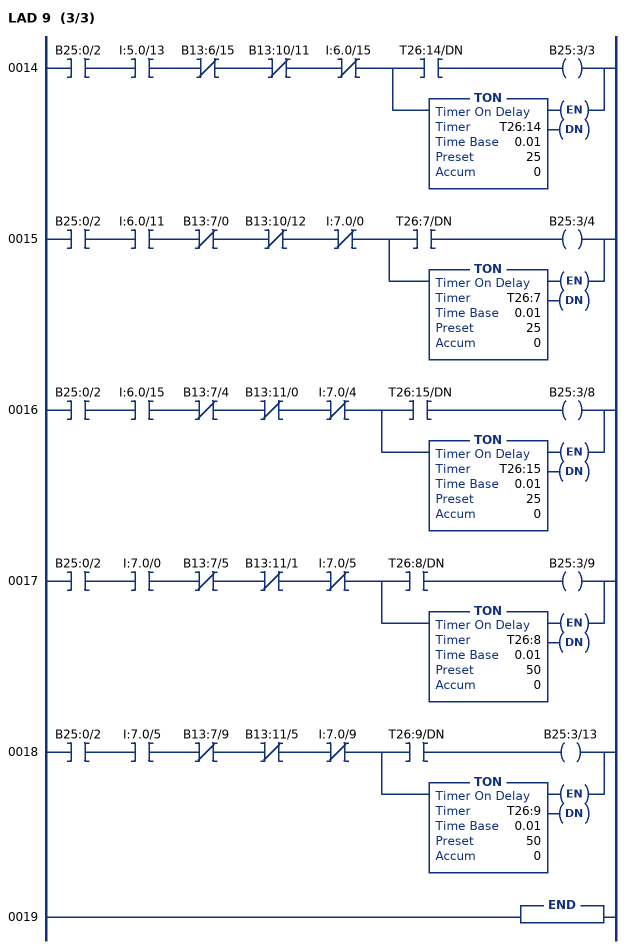
% Rung: 14 %
SOR XIC B25:0/2 XIC I:5.0/13 XIO B13:6/15 XIO B13:10/11 XIO I:6.0/15 BST XIC T26:14/DN OTE B25:3/3 NXB TON T26:14 0.01 25 0 BND EOR
% Rung: 15 %
SOR XIC B25:0/2 XIC I:6.0/11 XIO B13:7/0 XIO B13:10/12 XIO I:7.0/0 BST XIC T26:7/DN OTE B25:3/4 NXB TON T26:7 0.01 25 0 BND EOR
% Rung: 16 %
SOR XIC B25:0/2 XIC I:6.0/15 XIO B13:7/4 XIO B13:11/0 XIO I:7.0/4 BST XIC T26:15/DN OTE B25:3/8 NXB TON T26:15 0.01 25 0 BND EOR
% Rung: 17 %
SOR XIC B25:0/2 XIC I:7.0/0 XIO B13:7/5 XIO B13:11/1 XIO I:7.0/5 BST XIC T26:8/DN OTE B25:3/9 NXB TON T26:8 0.01 50 0 BND EOR
% Rung: 18 %
SOR XIC B25:0/2 XIC I:7.0/5 XIO B13:7/9 XIO B13:11/5 XIO I:7.0/9 BST XIC T26:9/DN OTE B25:3/13 NXB TON T26:9 0.01 50 0 BND EOR
% Rung: 19 %
SOR END EOR

LADDER 10
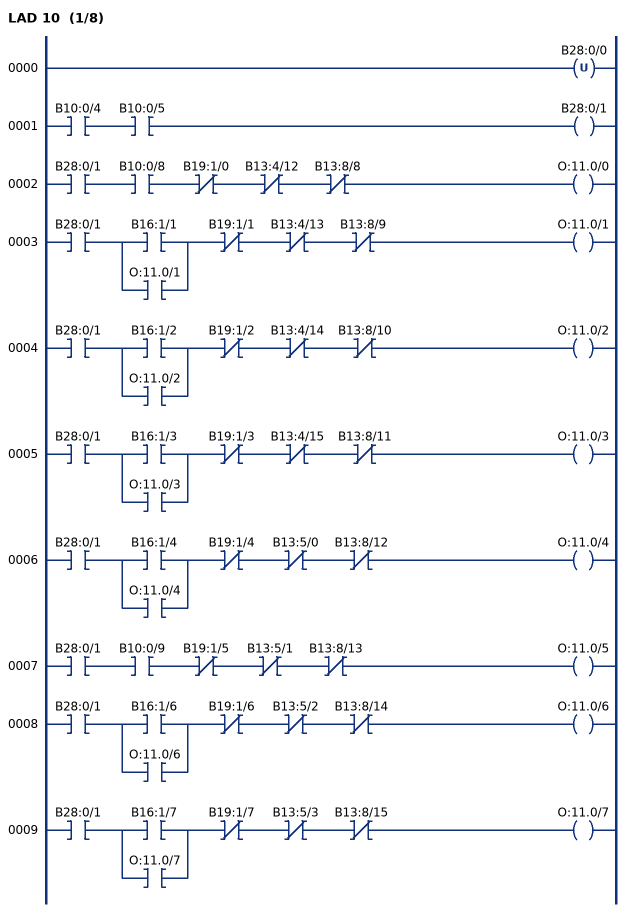
% Rung: 0 %
SOR OTU B28:0/0 EOR
% Rung: 1 %
SOR XIC B10:0/4 XIC B10:0/5 OTE B28:0/1 EOR
% Rung: 2 %
SOR XIC B28:0/1 XIC B10:0/8 XIO B19:1/0 XIO B13:4/12 XIO B13:8/8 OTE O:11.0/0 EOR
% Rung: 3 %
SOR XIC B28:0/1 BST XIC B16:1/1 NXB XIC O:11.0/1 BND XIO B19:1/1 XIO B13:4/13 XIO B13:8/9 OTE O:11.0/1 EOR
% Rung: 4 %
SOR XIC B28:0/1 BST XIC B16:1/2 NXB XIC O:11.0/2 BND XIO B19:1/2 XIO B13:4/14 XIO B13:8/10 OTE O:11.0/2 EOR
% Rung: 5 %
SOR XIC B28:0/1 BST XIC B16:1/3 NXB XIC O:11.0/3 BND XIO B19:1/3 XIO B13:4/15 XIO B13:8/11 OTE O:11.0/3 EOR
% Rung: 6 %
SOR XIC B28:0/1 BST XIC B16:1/4 NXB XIC O:11.0/4 BND XIO B19:1/4 XIO B13:5/0 XIO B13:8/12 OTE O:11.0/4 EOR
% Rung: 7 %
SOR XIC B28:0/1 XIC B10:0/9 XIO B19:1/5 XIO B13:5/1 XIO B13:8/13 OTE O:11.0/5 EOR
% Rung: 8 %
SOR XIC B28:0/1 BST XIC B16:1/6 NXB XIC O:11.0/6 BND XIO B19:1/6 XIO B13:5/2 XIO B13:8/14 OTE O:11.0/6 EOR
% Rung: 9 %
SOR XIC B28:0/1 BST XIC B16:1/7 NXB XIC O:11.0/7 BND XIO B19:1/7 XIO B13:5/3 XIO B13:8/15 OTE O:11.0/7 EOR

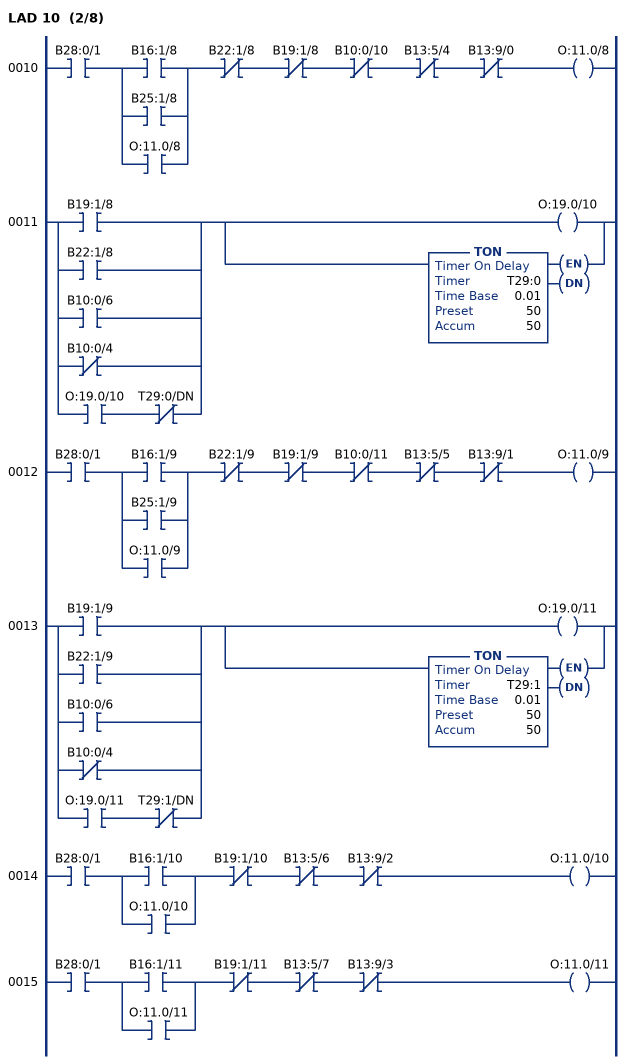
% Rung: 10 %
SOR XIC B28:0/1 BST XIC B16:1/8 NXB XIC B25:1/8 NXB XIC O:11.0/8 BND XIO B22:1/8 XIO B19:1/8 XIO B10:0/10 XIO B13:5/4 XIO B13:9/0 OTE O:11.0/8 EOR
% Rung: 11 %
SOR BST XIC B19:1/8 NXB XIC B22:1/8 NXB XIC B10:0/6 NXB XIO B10:0/4 NXB XIC O:19.0/10 XIO T29:0/DN BND BST OTE O:19.0/10 NXB TON T29:0 0.01 50 50 BND EOR
% Rung: 12 %
SOR XIC B28:0/1 BST XIC B16:1/9 NXB XIC B25:1/9 NXB XIC O:11.0/9 BND XIO B22:1/9 XIO B19:1/9 XIO B10:0/11 XIO B13:5/5 XIO B13:9/1 OTE O:11.0/9 EOR
% Rung: 13 %
SOR BST XIC B19:1/9 NXB XIC B22:1/9 NXB XIC B10:0/6 NXB XIO B10:0/4 NXB XIC O:19.0/11 XIO T29:1/DN BND BST OTE O:19.0/11 NXB TON T29:1 0.01 50 50 BND EOR
% Rung: 14 %
SOR XIC B28:0/1 BST XIC B16:1/10 NXB XIC O:11.0/10 BND XIO B19:1/10 XIO B13:5/6 XIO B13:9/2 OTE O:11.0/10 EOR
% Rung: 15 %
SOR XIC B28:0/1 BST XIC B16:1/11 NXB XIC O:11.0/11 BND XIO B19:1/11 XIO B13:5/7 XIO B13:9/3 OTE O:11.0/11 EOR

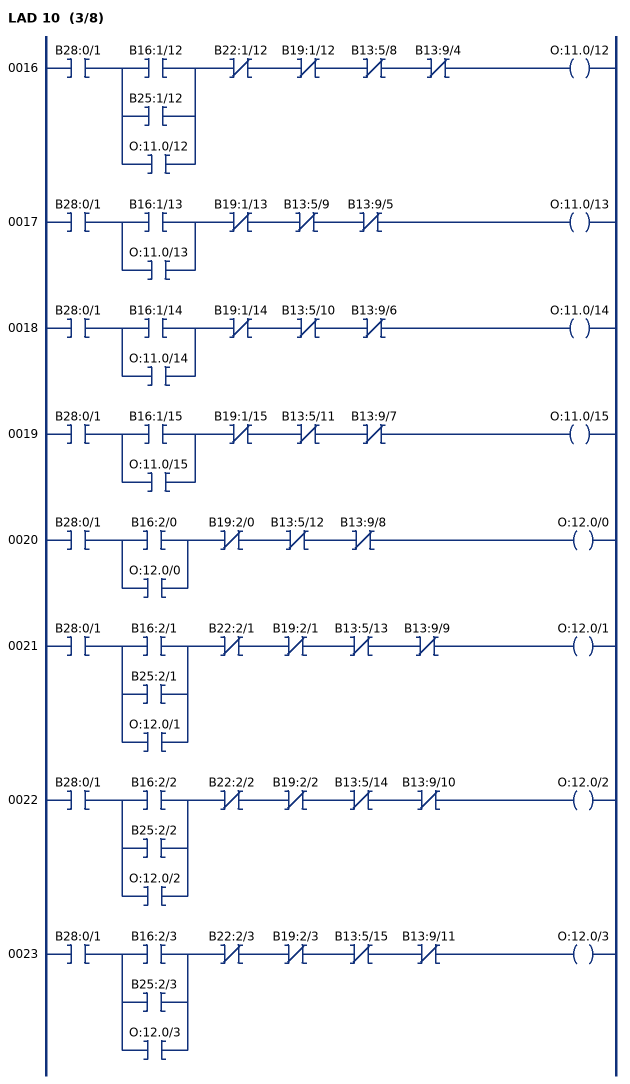
% Rung: 16 %
SOR XIC B28:0/1 BST XIC B16:1/12 NXB XIC B25:1/12 NXB XIC O:11.0/12 BND XIO B22:1/12 XIO B19:1/12 XIO B13:5/8 XIO B13:9/4 OTE O:11.0/12 EOR
% Rung: 17 %
SOR XIC B28:0/1 BST XIC B16:1/13 NXB XIC O:11.0/13 BND XIO B19:1/13 XIO B13:5/9 XIO B13:9/5 OTE O:11.0/13 EOR
% Rung: 18 %
SOR XIC B28:0/1 BST XIC B16:1/14 NXB XIC O:11.0/14 BND XIO B19:1/14 XIO B13:5/10 XIO B13:9/6 OTE O:11.0/14 EOR
% Rung: 19 %
SOR XIC B28:0/1 BST XIC B16:1/15 NXB XIC O:11.0/15 BND XIO B19:1/15 XIO B13:5/11 XIO B13:9/7 OTE O:11.0/15 EOR
% Rung: 20 %
SOR XIC B28:0/1 BST XIC B16:2/0 NXB XIC O:12.0/0 BND XIO B19:2/0 XIO B13:5/12 XIO B13:9/8 OTE O:12.0/0 EOR
% Rung: 21 %
SOR XIC B28:0/1 BST XIC B16:2/1 NXB XIC B25:2/1 NXB XIC O:12.0/1 BND XIO B22:2/1 XIO B19:2/1 XIO B13:5/13 XIO B13:9/9 OTE O:12.0/1 EOR
% Rung: 22 %
SOR XIC B28:0/1 BST XIC B16:2/2 NXB XIC B25:2/2 NXB XIC O:12.0/2 BND XIO B22:2/2 XIO B19:2/2 XIO B13:5/14 XIO B13:9/10 OTE O:12.0/2 EOR
% Rung: 23 %
SOR XIC B28:0/1 BST XIC B16:2/3 NXB XIC B25:2/3 NXB XIC O:12.0/3 BND XIO B22:2/3 XIO B19:2/3 XIO B13:5/15 XIO B13:9/11 OTE O:12.0/3 EOR

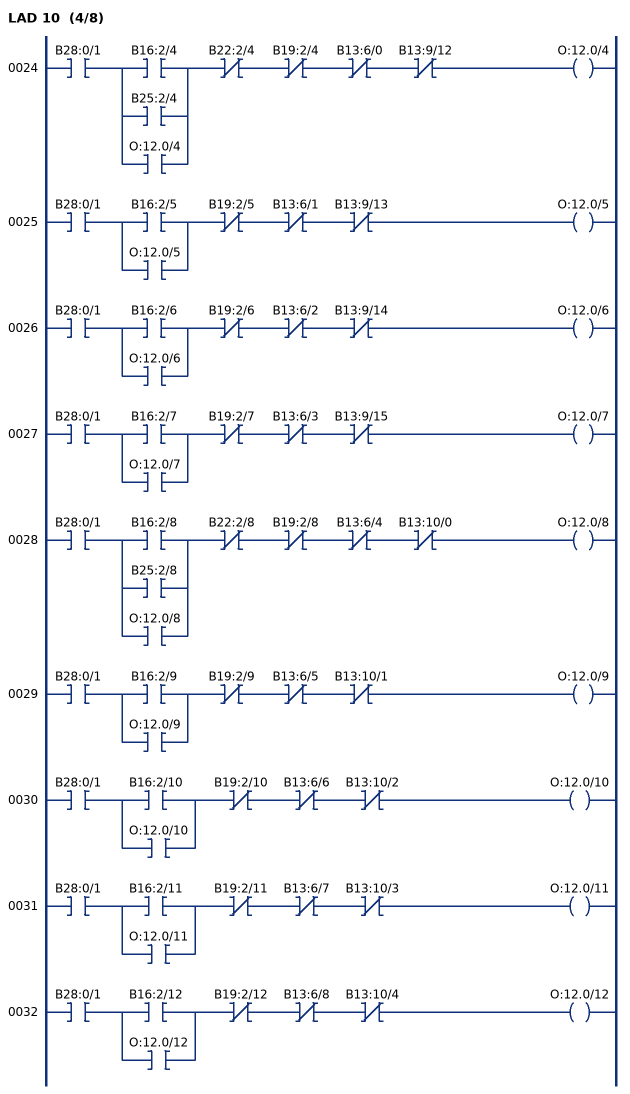
% Rung: 24 %
SOR XIC B28:0/1 BST XIC B16:2/4 NXB XIC B25:2/4 NXB XIC O:12.0/4 BND XIO B22:2/4 XIO B19:2/4 XIO B13:6/0 XIO B13:9/12 OTE O:12.0/4 EOR
% Rung: 25 %
SOR XIC B28:0/1 BST XIC B16:2/5 NXB XIC O:12.0/5 BND XIO B19:2/5 XIO B13:6/1 XIO B13:9/13 OTE O:12.0/5 EOR
% Rung: 26 %
SOR XIC B28:0/1 BST XIC B16:2/6 NXB XIC O:12.0/6 BND XIO B19:2/6 XIO B13:6/2 XIO B13:9/14 OTE O:12.0/6 EOR
% Rung: 27 %
SOR XIC B28:0/1 BST XIC B16:2/7 NXB XIC O:12.0/7 BND XIO B19:2/7 XIO B13:6/3 XIO B13:9/15 OTE O:12.0/7 EOR
% Rung: 28 %
SOR XIC B28:0/1 BST XIC B16:2/8 NXB XIC B25:2/8 NXB XIC O:12.0/8 BND XIO B22:2/8 XIO B19:2/8 XIO B13:6/4 XIO B13:10/0 OTE O:12.0/8 EOR
% Rung: 29 %
SOR XIC B28:0/1 BST XIC B16:2/9 NXB XIC O:12.0/9 BND XIO B19:2/9 XIO B13:6/5 XIO B13:10/1 OTE O:12.0/9 EOR
% Rung: 30 %
SOR XIC B28:0/1 BST XIC B16:2/10 NXB XIC O:12.0/10 BND XIO B19:2/10 XIO B13:6/6 XIO B13:10/2 OTE O:12.0/10 EOR
% Rung: 31 %
SOR XIC B28:0/1 BST XIC B16:2/11 NXB XIC O:12.0/11 BND XIO B19:2/11 XIO B13:6/7 XIO B13:10/3 OTE O:12.0/11 EOR
% Rung: 32 %
SOR XIC B28:0/1 BST XIC B16:2/12 NXB XIC O:12.0/12 BND XIO B19:2/12 XIO B13:6/8 XIO B13:10/4 OTE O:12.0/12 EOR

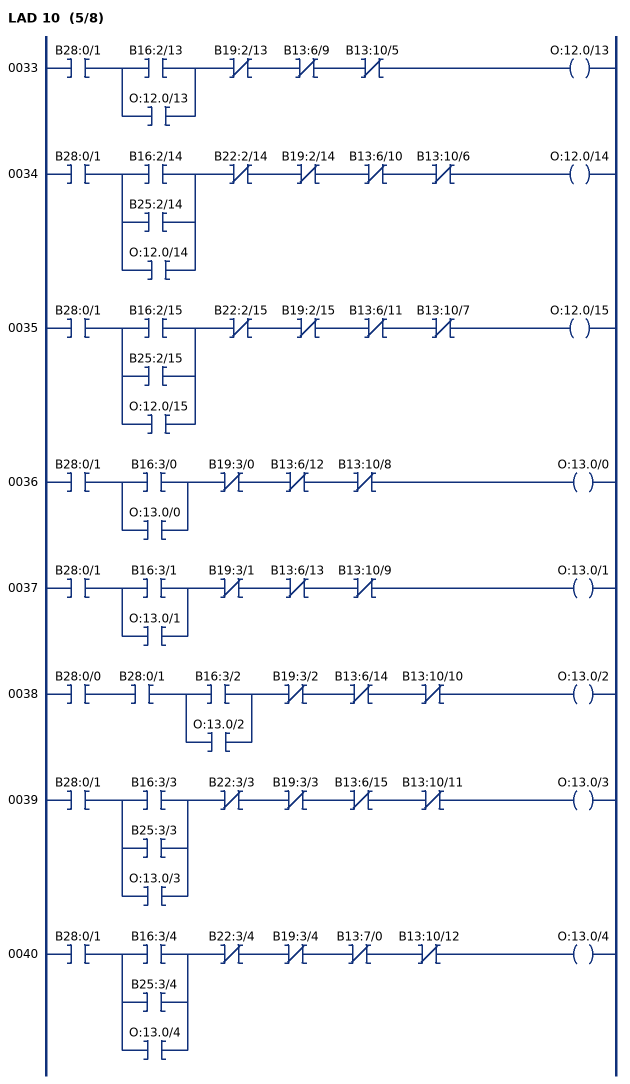
% Rung: 33 %
SOR XIC B28:0/1 BST XIC B16:2/13 NXB XIC O:12.0/13 BND XIO B19:2/13 XIO B13:6/9 XIO B13:10/5 OTE O:12.0/13 EOR
% Rung: 34 %
SOR XIC B28:0/1 BST XIC B16:2/14 NXB XIC B25:2/14 NXB XIC O:12.0/14 BND XIO B22:2/14 XIO B19:2/14 XIO B13:6/10 XIO B13:10/6 OTE O:12.0/14 EOR
% Rung: 35 %
SOR XIC B28:0/1 BST XIC B16:2/15 NXB XIC B25:2/15 NXB XIC O:12.0/15 BND XIO B22:2/15 XIO B19:2/15 XIO B13:6/11 XIO B13:10/7 OTE O:12.0/15 EOR
% Rung: 36 %
SOR XIC B28:0/1 BST XIC B16:3/0 NXB XIC O:13.0/0 BND XIO B19:3/0 XIO B13:6/12 XIO B13:10/8 OTE O:13.0/0 EOR
% Rung: 37 %
SOR XIC B28:0/1 BST XIC B16:3/1 NXB XIC O:13.0/1 BND XIO B19:3/1 XIO B13:6/13 XIO B13:10/9 OTE O:13.0/1 EOR
% Rung: 38 %
SOR XIC B28:0/0 XIC B28:0/1 BST XIC B16:3/2 NXB XIC O:13.0/2 BND XIO B19:3/2 XIO B13:6/14 XIO B13:10/10 OTE O:13.0/2 EOR
% Rung: 39 %
SOR XIC B28:0/1 BST XIC B16:3/3 NXB XIC B25:3/3 NXB XIC O:13.0/3 BND XIO B22:3/3 XIO B19:3/3 XIO B13:6/15 XIO B13:10/11 OTE O:13.0/3 EOR
% Rung: 40 %
SOR XIC B28:0/1 BST XIC B16:3/4 NXB XIC B25:3/4 NXB XIC O:13.0/4 BND XIO B22:3/4 XIO B19:3/4 XIO B13:7/0 XIO B13:10/12 OTE O:13.0/4 EOR

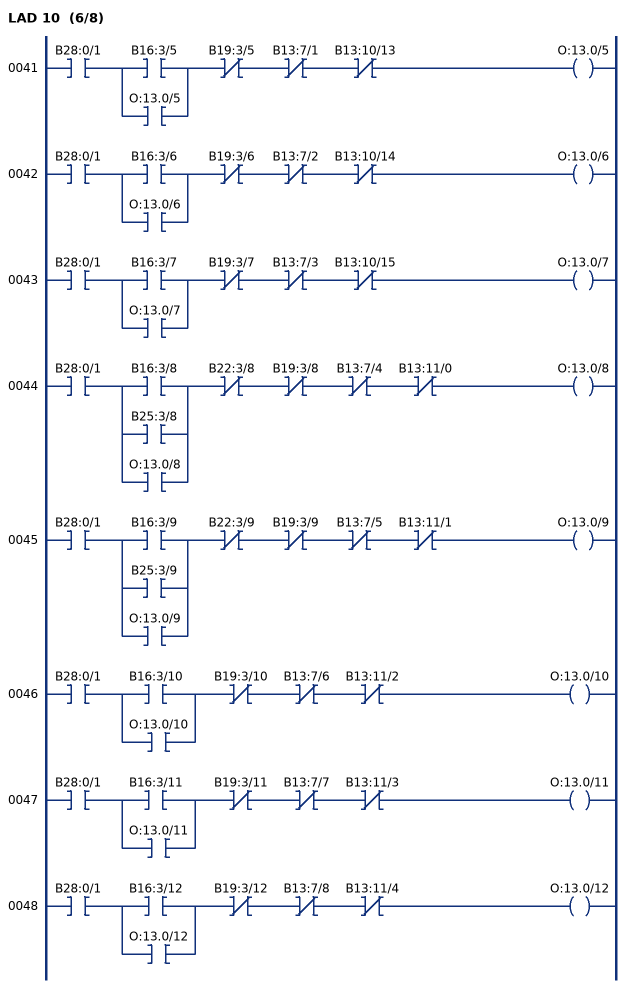
% Rung: 41 %
SOR XIC B28:0/1 BST XIC B16:3/5 NXB XIC O:13.0/5 BND XIO B19:3/5 XIO B13:7/1 XIO B13:10/13 OTE O:13.0/5 EOR
% Rung: 42 %
SOR XIC B28:0/1 BST XIC B16:3/6 NXB XIC O:13.0/6 BND XIO B19:3/6 XIO B13:7/2 XIO B13:10/14 OTE O:13.0/6 EOR
% Rung: 43 %
SOR XIC B28:0/1 BST XIC B16:3/7 NXB XIC O:13.0/7 BND XIO B19:3/7 XIO B13:7/3 XIO B13:10/15 OTE O:13.0/7 EOR
% Rung: 44 %
SOR XIC B28:0/1 BST XIC B16:3/8 NXB XIC B25:3/8 NXB XIC O:13.0/8 BND XIO B22:3/8 XIO B19:3/8 XIO B13:7/4 XIO B13:11/0 OTE O:13.0/8 EOR
% Rung: 45 %
SOR XIC B28:0/1 BST XIC B16:3/9 NXB XIC B25:3/9 NXB XIC O:13.0/9 BND XIO B22:3/9 XIO B19:3/9 XIO B13:7/5 XIO B13:11/1 OTE O:13.0/9 EOR
% Rung: 46 %
SOR XIC B28:0/1 BST XIC B16:3/10 NXB XIC O:13.0/10 BND XIO B19:3/10 XIO B13:7/6 XIO B13:11/2 OTE O:13.0/10 EOR
% Rung: 47 %
SOR XIC B28:0/1 BST XIC B16:3/11 NXB XIC O:13.0/11 BND XIO B19:3/11 XIO B13:7/7 XIO B13:11/3 OTE O:13.0/11 EOR
% Rung: 48 %
SOR XIC B28:0/1 BST XIC B16:3/12 NXB XIC O:13.0/12 BND XIO B19:3/12 XIO B13:7/8 XIO B13:11/4 OTE O:13.0/12 EOR

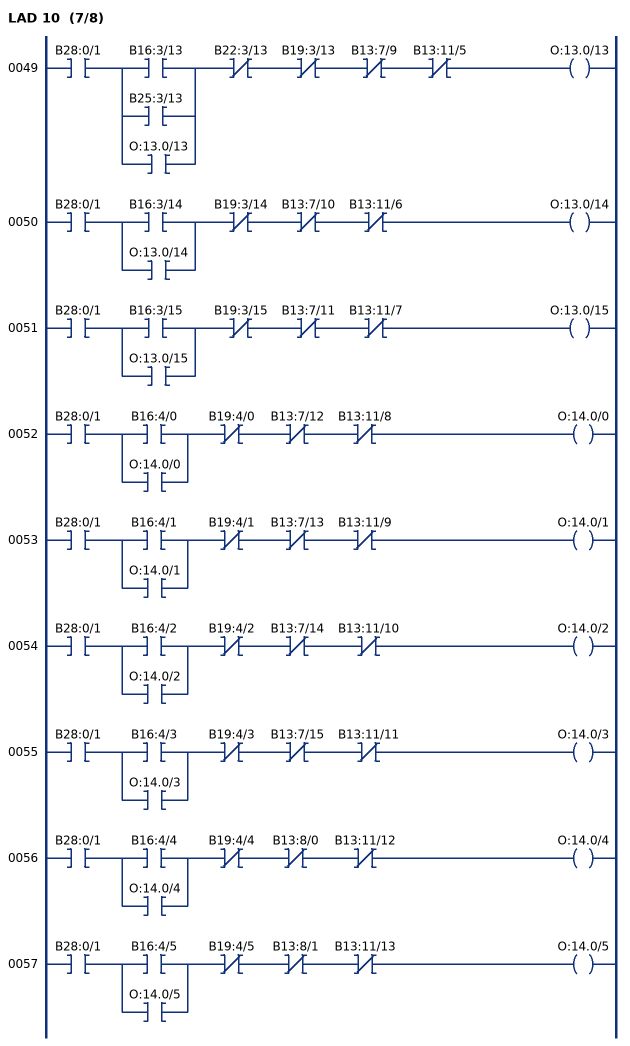
% Rung: 49 %
SOR XIC B28:0/1 BST XIC B16:3/13 NXB XIC B25:3/13 NXB XIC O:13.0/13 BND XIO B22:3/13 XIO B19:3/13 XIO B13:7/9 XIO B13:11/5 OTE O:13.0/13 EOR
% Rung: 50 %
SOR XIC B28:0/1 BST XIC B16:3/14 NXB XIC O:13.0/14 BND XIO B19:3/14 XIO B13:7/10 XIO B13:11/6 OTE O:13.0/14 EOR
% Rung: 51 %
SOR XIC B28:0/1 BST XIC B16:3/15 NXB XIC O:13.0/15 BND XIO B19:3/15 XIO B13:7/11 XIO B13:11/7 OTE O:13.0/15 EOR
% Rung: 52 %
SOR XIC B28:0/1 BST XIC B16:4/0 NXB XIC O:14.0/0 BND XIO B19:4/0 XIO B13:7/12 XIO B13:11/8 OTE O:14.0/0 EOR
% Rung: 53 %
SOR XIC B28:0/1 BST XIC B16:4/1 NXB XIC O:14.0/1 BND XIO B19:4/1 XIO B13:7/13 XIO B13:11/9 OTE O:14.0/1 EOR
% Rung: 54 %
SOR XIC B28:0/1 BST XIC B16:4/2 NXB XIC O:14.0/2 BND XIO B19:4/2 XIO B13:7/14 XIO B13:11/10 OTE O:14.0/2 EOR
% Rung: 55 %
SOR XIC B28:0/1 BST XIC B16:4/3 NXB XIC O:14.0/3 BND XIO B19:4/3 XIO B13:7/15 XIO B13:11/11 OTE O:14.0/3 EOR
% Rung: 56 %
SOR XIC B28:0/1 BST XIC B16:4/4 NXB XIC O:14.0/4 BND XIO B19:4/4 XIO B13:8/0 XIO B13:11/12 OTE O:14.0/4 EOR
% Rung: 57 %
SOR XIC B28:0/1 BST XIC B16:4/5 NXB XIC O:14.0/5 BND XIO B19:4/5 XIO B13:8/1 XIO B13:11/13 OTE O:14.0/5 EOR

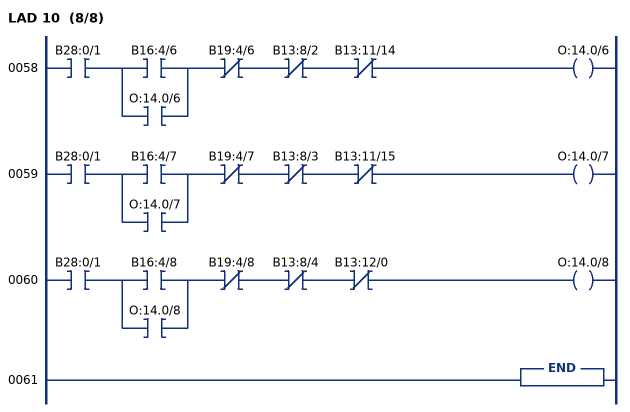
% Rung: 58 %
SOR XIC B28:0/1 BST XIC B16:4/6 NXB XIC O:14.0/6 BND XIO B19:4/6 XIO B13:8/2 XIO B13:11/14 OTE O:14.0/6 EOR
% Rung: 59 %
SOR XIC B28:0/1 BST XIC B16:4/7 NXB XIC O:14.0/7 BND XIO B19:4/7 XIO B13:8/3 XIO B13:11/15 OTE O:14.0/7 EOR
% Rung: 60 %
SOR XIC B28:0/1 BST XIC B16:4/8 NXB XIC O:14.0/8 BND XIO B19:4/8 XIO B13:8/4 XIO B13:12/0 OTE O:14.0/8 EOR
% Rung: 61 %
SOR END EOR

LADDER 11
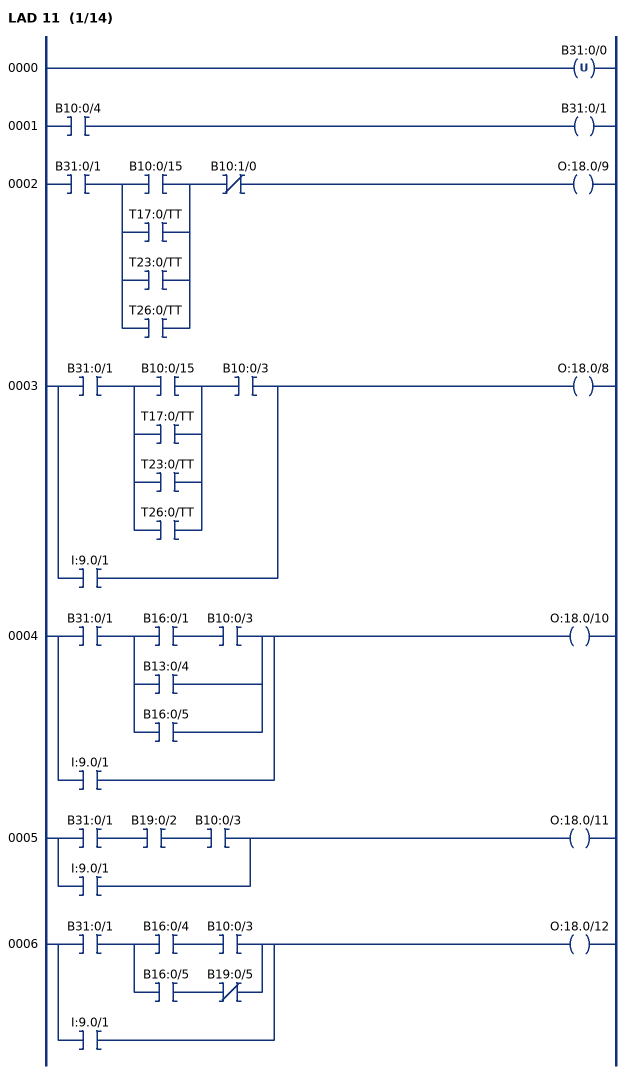
% Rung: 0 %
SOR OTU B31:0/0 EOR
% Rung: 1 %
SOR XIC B10:0/4 OTE B31:0/1 EOR
% Rung: 2 %
SOR XIC B31:0/1 BST XIC B10:0/15 NXB XIC T17:0/TT NXB XIC T23:0/TT NXB XIC T26:0/TT BND XIO B10:1/0 OTE O:18.0/9 EOR
% Rung: 3 %
SOR BST XIC B31:0/1 BST XIC B10:0/15 NXB XIC T17:0/TT NXB XIC T23:0/TT NXB XIC T26:0/TT BND XIC B10:0/3 NXB XIC I:9.0/1 BND OTE O:18.0/8 EOR
% Rung: 4 %
SOR BST XIC B31:0/1 BST XIC B16:0/1 XIC B10:0/3 NXB XIC B13:0/4 NXB XIC B16:0/5 BND NXB XIC I:9.0/1 BND OTE O:18.0/10 EOR
% Rung: 5 %
SOR BST XIC B31:0/1 XIC B19:0/2 XIC B10:0/3 NXB XIC I:9.0/1 BND OTE O:18.0/11 EOR
% Rung: 6 %
SOR BST XIC B31:0/1 BST XIC B16:0/4 XIC B10:0/3 NXB XIC B16:0/5 XIO B19:0/5 BND NXB XIC I:9.0/1 BND OTE O:18.0/12 EOR

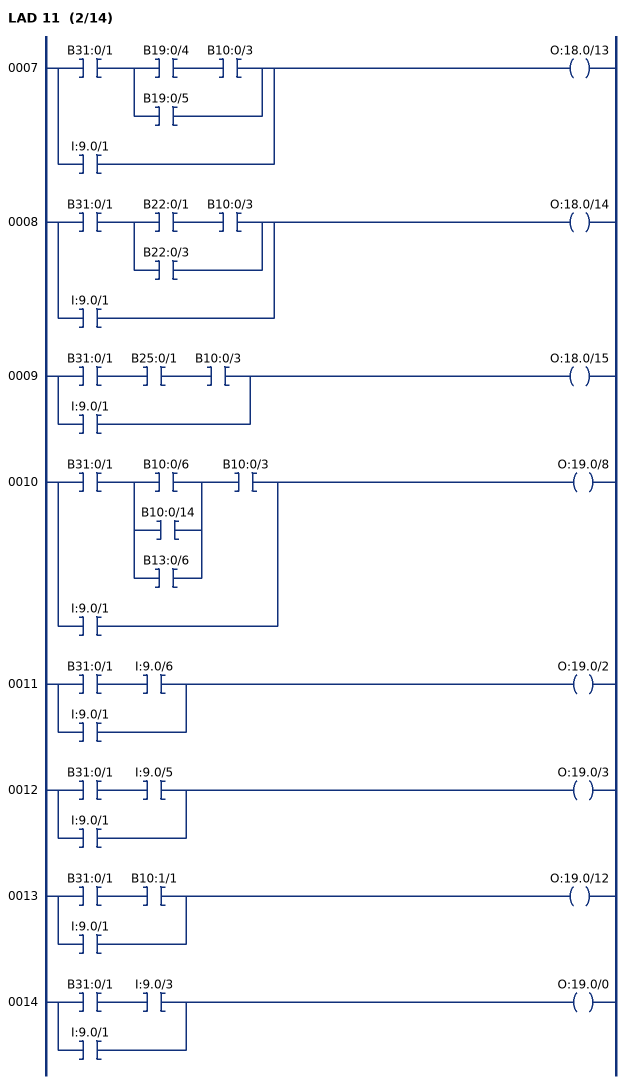
% Rung: 7 %
SOR BST XIC B31:0/1 BST XIC B19:0/4 XIC B10:0/3 NXB XIC B19:0/5 BND NXB XIC I:9.0/1 BND OTE O:18.0/13 EOR
% Rung: 8 %
SOR BST XIC B31:0/1 BST XIC B22:0/1 XIC B10:0/3 NXB XIC B22:0/3 BND NXB XIC I:9.0/1 BND OTE O:18.0/14 EOR
% Rung: 9 %
SOR BST XIC B31:0/1 XIC B25:0/1 XIC B10:0/3 NXB XIC I:9.0/1 BND OTE O:18.0/15 EOR
% Rung: 10 %
SOR BST XIC B31:0/1 BST XIC B10:0/6 NXB XIC B10:0/14 NXB XIC B13:0/6 BND XIC B10:0/3 NXB XIC I:9.0/1 BND OTE O:19.0/8 EOR
% Rung: 11 %
SOR BST XIC B31:0/1 XIC I:9.0/6 NXB XIC I:9.0/1 BND OTE O:19.0/2 EOR
% Rung: 12 %
SOR BST XIC B31:0/1 XIC I:9.0/5 NXB XIC I:9.0/1 BND OTE O:19.0/3 EOR
% Rung: 13 %
SOR BST XIC B31:0/1 XIC B10:1/1 NXB XIC I:9.0/1 BND OTE O:19.0/12 EOR
% Rung: 14 %
SOR BST XIC B31:0/1 XIC I:9.0/3 NXB XIC I:9.0/1 BND OTE O:19.0/0 EOR

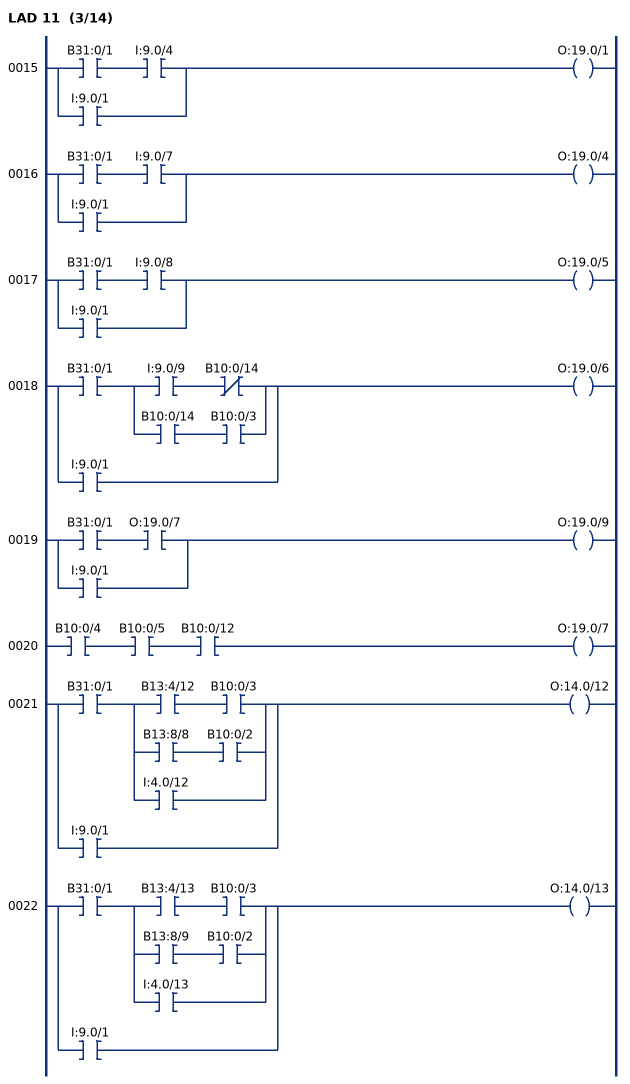
% Rung: 15 %
SOR BST XIC B31:0/1 XIC I:9.0/4 NXB XIC I:9.0/1 BND OTE O:19.0/1 EOR
% Rung: 16 %
SOR BST XIC B31:0/1 XIC I:9.0/7 NXB XIC I:9.0/1 BND OTE O:19.0/4 EOR
% Rung: 17 %
SOR BST XIC B31:0/1 XIC I:9.0/8 NXB XIC I:9.0/1 BND OTE O:19.0/5 EOR
% Rung: 18 %
SOR BST XIC B31:0/1 BST XIC I:9.0/9 XIO B10:0/14 NXB XIC B10:0/14 XIC B10:0/3 BND NXB XIC I:9.0/1 BND OTE O:19.0/6 EOR
% Rung: 19 %
SOR BST XIC B31:0/1 XIC O:19.0/7 NXB XIC I:9.0/1 BND OTE O:19.0/9 EOR
% Rung: 20 %
SOR XIC B10:0/4 XIC B10:0/5 XIC B10:0/12 OTE O:19.0/7 EOR
% Rung: 21 %
SOR BST XIC B31:0/1 BST XIC B13:4/12 XIC B10:0/3 NXB XIC B13:8/8 XIC B10:0/2 NXB XIC I:4.0/12 BND NXB XIC I:9.0/1 BND OTE O:14.0/12 EOR
% Rung: 22 %
SOR BST XIC B31:0/1 BST XIC B13:4/13 XIC B10:0/3 NXB XIC B13:8/9 XIC B10:0/2 NXB XIC I:4.0/13 BND NXB XIC I:9.0/1 BND OTE O:14.0/13 EOR

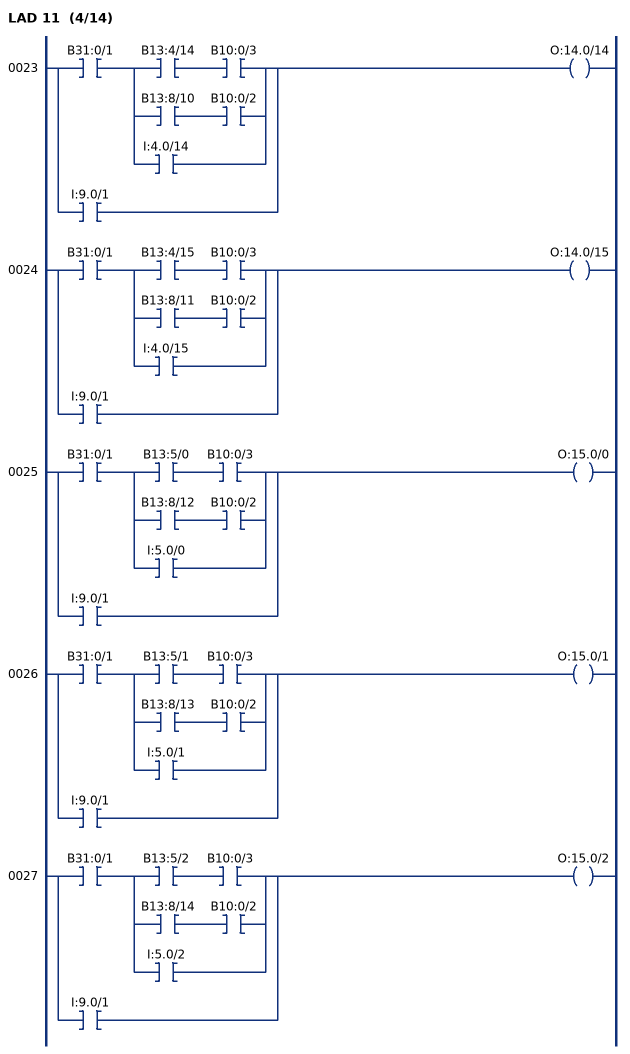
% Rung: 23 %
SOR BST XIC B31:0/1 BST XIC B13:4/14 XIC B10:0/3 NXB XIC B13:8/10 XIC B10:0/2 NXB XIC I:4.0/14 BND NXB XIC I:9.0/1 BND OTE O:14.0/14 EOR
% Rung: 24 %
SOR BST XIC B31:0/1 BST XIC B13:4/15 XIC B10:0/3 NXB XIC B13:8/11 XIC B10:0/2 NXB XIC I:4.0/15 BND NXB XIC I:9.0/1 BND OTE O:14.0/15 EOR
% Rung: 25 %
SOR BST XIC B31:0/1 BST XIC B13:5/0 XIC B10:0/3 NXB XIC B13:8/12 XIC B10:0/2 NXB XIC I:5.0/0 BND NXB XIC I:9.0/1 BND OTE O:15.0/0 EOR
% Rung: 26 %
SOR BST XIC B31:0/1 BST XIC B13:5/1 XIC B10:0/3 NXB XIC B13:8/13 XIC B10:0/2 NXB XIC I:5.0/1 BND NXB XIC I:9.0/1 BND OTE O:15.0/1 EOR
% Rung: 27 %
SOR BST XIC B31:0/1 BST XIC B13:5/2 XIC B10:0/3 NXB XIC B13:8/14 XIC B10:0/2 NXB XIC I:5.0/2 BND NXB XIC I:9.0/1 BND OTE O:15.0/2 EOR

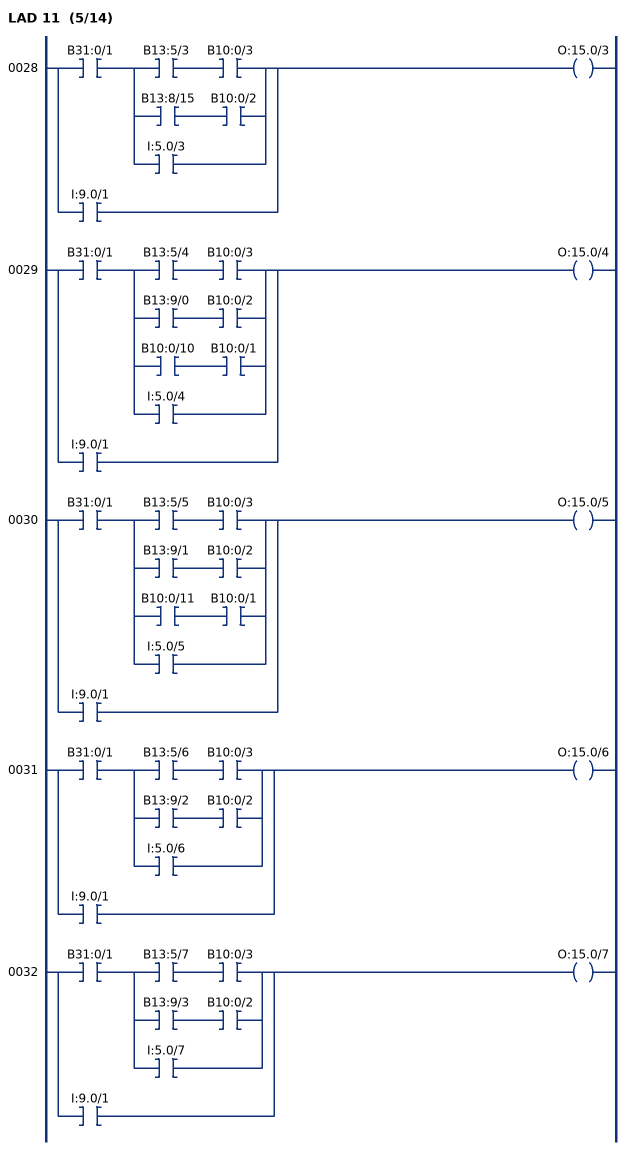
% Rung: 28 %
SOR BST XIC B31:0/1 BST XIC B13:5/3 XIC B10:0/3 NXB XIC B13:8/15 XIC B10:0/2 NXB XIC I:5.0/3 BND NXB XIC I:9.0/1 BND OTE O:15.0/3 EOR
% Rung: 29 %
SOR BST XIC B31:0/1 BST XIC B13:5/4 XIC B10:0/3 NXB XIC B13:9/0 XIC B10:0/2 NXB XIC B10:0/10 XIC B10:0/1 NXB XIC I:5.0/4 BND NXB XIC I:9.0/1 BND OTE O:15.0/4 EOR
% Rung: 30 %
SOR BST XIC B31:0/1 BST XIC B13:5/5 XIC B10:0/3 NXB XIC B13:9/1 XIC B10:0/2 NXB XIC B10:0/11 XIC B10:0/1 NXB XIC I:5.0/5 BND NXB XIC I:9.0/1 BND OTE O:15.0/5 EOR
% Rung: 31 %
SOR BST XIC B31:0/1 BST XIC B13:5/6 XIC B10:0/3 NXB XIC B13:9/2 XIC B10:0/2 NXB XIC I:5.0/6 BND NXB XIC I:9.0/1 BND OTE O:15.0/6 EOR
% Rung: 32 %
SOR BST XIC B31:0/1 BST XIC B13:5/7 XIC B10:0/3 NXB XIC B13:9/3 XIC B10:0/2 NXB XIC I:5.0/7 BND NXB XIC I:9.0/1 BND OTE O:15.0/7 EOR

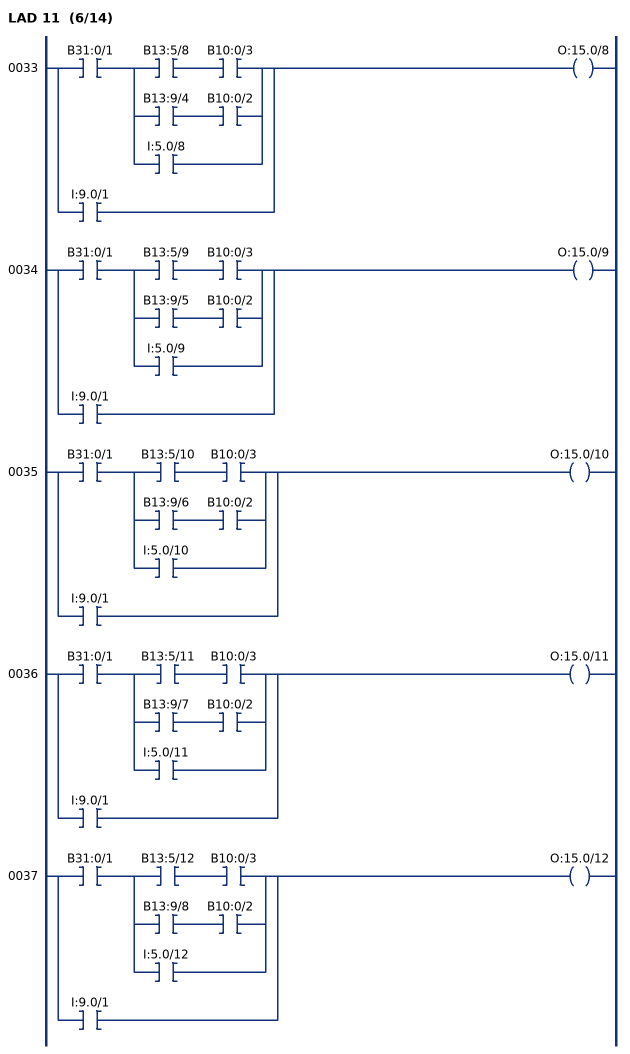
% Rung: 33 %
SOR BST XIC B31:0/1 BST XIC B13:5/8 XIC B10:0/3 NXB XIC B13:9/4 XIC B10:0/2 NXB XIC I:5.0/8 BND NXB XIC I:9.0/1 BND OTE O:15.0/8 EOR
% Rung: 34 %
SOR BST XIC B31:0/1 BST XIC B13:5/9 XIC B10:0/3 NXB XIC B13:9/5 XIC B10:0/2 NXB XIC I:5.0/9 BND NXB XIC I:9.0/1 BND OTE O:15.0/9 EOR
% Rung: 35 %
SOR BST XIC B31:0/1 BST XIC B13:5/10 XIC B10:0/3 NXB XIC B13:9/6 XIC B10:0/2 NXB XIC I:5.0/10 BND NXB XIC I:9.0/1 BND OTE O:15.0/10 EOR
% Rung: 36 %
SOR BST XIC B31:0/1 BST XIC B13:5/11 XIC B10:0/3 NXB XIC B13:9/7 XIC B10:0/2 NXB XIC I:5.0/11 BND NXB XIC I:9.0/1 BND OTE O:15.0/11 EOR
% Rung: 37 %
SOR BST XIC B31:0/1 BST XIC B13:5/12 XIC B10:0/3 NXB XIC B13:9/8 XIC B10:0/2 NXB XIC I:5.0/12 BND NXB XIC I:9.0/1 BND OTE O:15.0/12 EOR

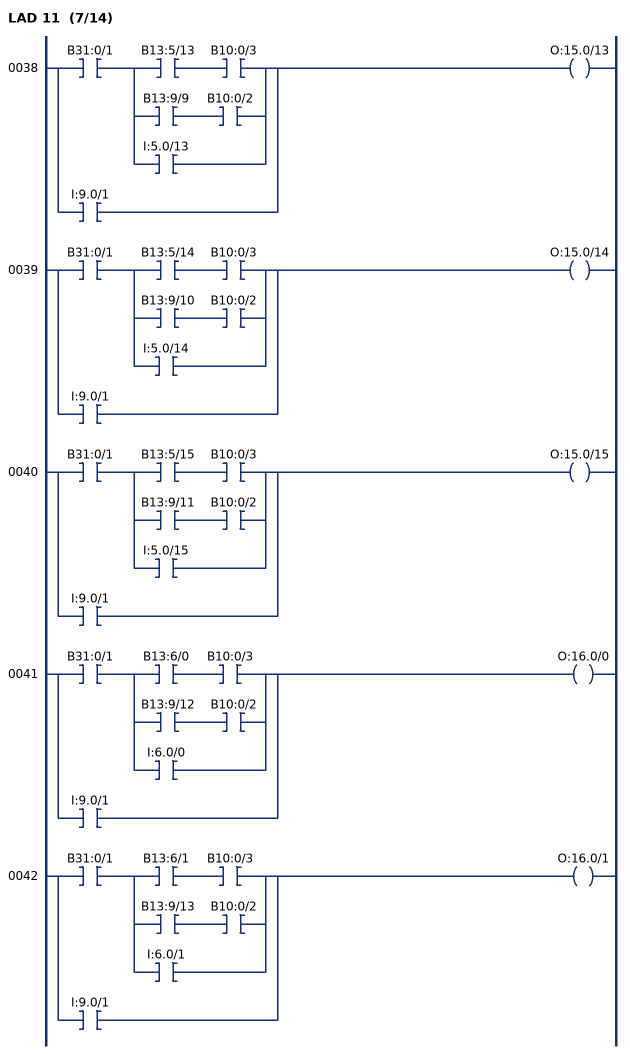
% Rung: 38 %
SOR BST XIC B31:0/1 BST XIC B13:5/13 XIC B10:0/3 NXB XIC B13:9/9 XIC B10:0/2 NXB XIC I:5.0/13 BND NXB XIC I:9.0/1 BND OTE O:15.0/13 EOR
% Rung: 39 %
SOR BST XIC B31:0/1 BST XIC B13:5/14 XIC B10:0/3 NXB XIC B13:9/10 XIC B10:0/2 NXB XIC I:5.0/14 BND NXB XIC I:9.0/1 BND OTE O:15.0/14 EOR
% Rung: 40 %
SOR BST XIC B31:0/1 BST XIC B13:5/15 XIC B10:0/3 NXB XIC B13:9/11 XIC B10:0/2 NXB XIC I:5.0/15 BND NXB XIC I:9.0/1 BND OTE O:15.0/15 EOR
% Rung: 41 %
SOR BST XIC B31:0/1 BST XIC B13:6/0 XIC B10:0/3 NXB XIC B13:9/12 XIC B10:0/2 NXB XIC I:6.0/0 BND NXB XIC I:9.0/1 BND OTE O:16.0/0 EOR
% Rung: 42 %
SOR BST XIC B31:0/1 BST XIC B13:6/1 XIC B10:0/3 NXB XIC B13:9/13 XIC B10:0/2 NXB XIC I:6.0/1 BND NXB XIC I:9.0/1 BND OTE O:16.0/1 EOR

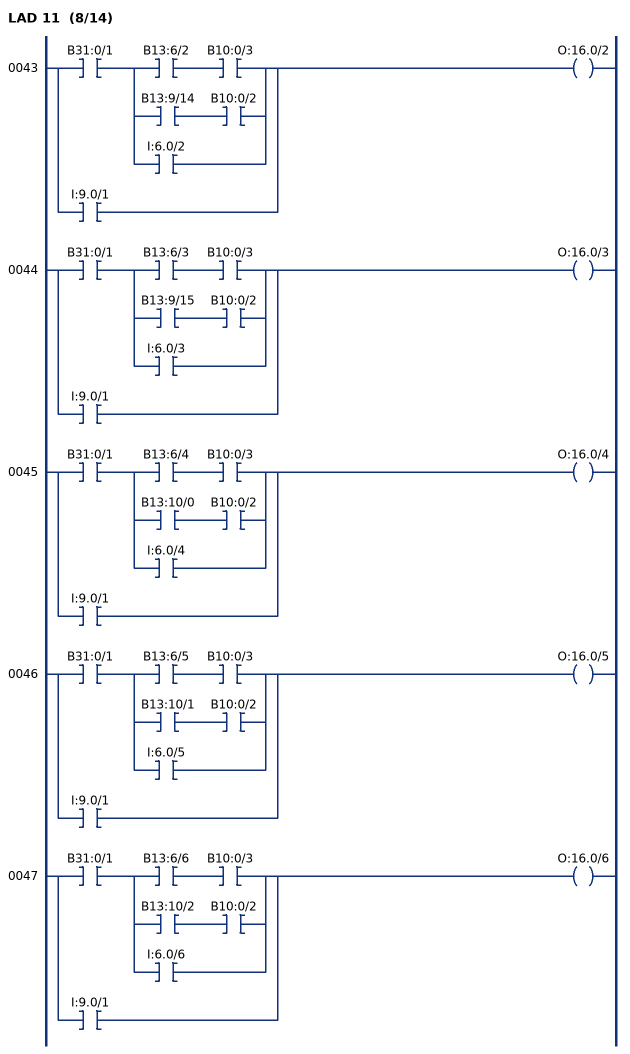
% Rung: 43 %
SOR BST XIC B31:0/1 BST XIC B13:6/2 XIC B10:0/3 NXB XIC B13:9/14 XIC B10:0/2 NXB XIC I:6.0/2 BND NXB XIC I:9.0/1 BND OTE O:16.0/2 EOR
% Rung: 44 %
SOR BST XIC B31:0/1 BST XIC B13:6/3 XIC B10:0/3 NXB XIC B13:9/15 XIC B10:0/2 NXB XIC I:6.0/3 BND NXB XIC I:9.0/1 BND OTE O:16.0/3 EOR
% Rung: 45 %
SOR BST XIC B31:0/1 BST XIC B13:6/4 XIC B10:0/3 NXB XIC B13:10/0 XIC B10:0/2 NXB XIC I:6.0/4 BND NXB XIC I:9.0/1 BND OTE O:16.0/4 EOR
% Rung: 46 %
SOR BST XIC B31:0/1 BST XIC B13:6/5 XIC B10:0/3 NXB XIC B13:10/1 XIC B10:0/2 NXB XIC I:6.0/5 BND NXB XIC I:9.0/1 BND OTE O:16.0/5 EOR
% Rung: 47 %
SOR BST XIC B31:0/1 BST XIC B13:6/6 XIC B10:0/3 NXB XIC B13:10/2 XIC B10:0/2 NXB XIC I:6.0/6 BND NXB XIC I:9.0/1 BND OTE O:16.0/6 EOR

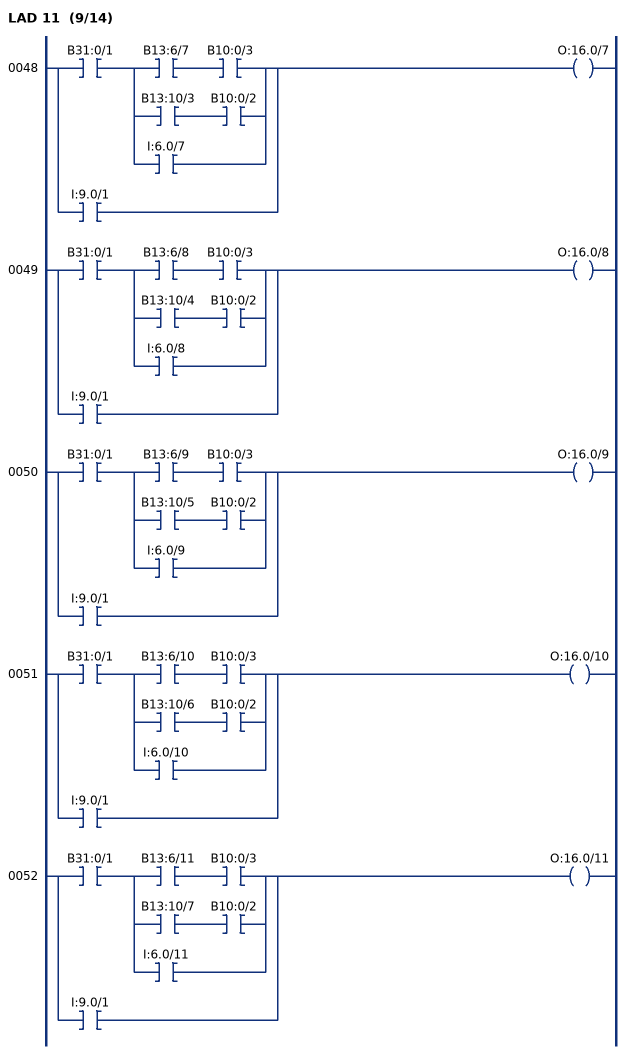
% Rung: 48 %
SOR BST XIC B31:0/1 BST XIC B13:6/7 XIC B10:0/3 NXB XIC B13:10/3 XIC B10:0/2 NXB XIC I:6.0/7 BND NXB XIC I:9.0/1 BND OTE O:16.0/7 EOR
% Rung: 49 %
SOR BST XIC B31:0/1 BST XIC B13:6/8 XIC B10:0/3 NXB XIC B13:10/4 XIC B10:0/2 NXB XIC I:6.0/8 BND NXB XIC I:9.0/1 BND OTE O:16.0/8 EOR
% Rung: 50 %
SOR BST XIC B31:0/1 BST XIC B13:6/9 XIC B10:0/3 NXB XIC B13:10/5 XIC B10:0/2 NXB XIC I:6.0/9 BND NXB XIC I:9.0/1 BND OTE O:16.0/9 EOR
% Rung: 51 %
SOR BST XIC B31:0/1 BST XIC B13:6/10 XIC B10:0/3 NXB XIC B13:10/6 XIC B10:0/2 NXB XIC I:6.0/10 BND NXB XIC I:9.0/1 BND OTE O:16.0/10 EOR
% Rung: 52 %
SOR BST XIC B31:0/1 BST XIC B13:6/11 XIC B10:0/3 NXB XIC B13:10/7 XIC B10:0/2 NXB XIC I:6.0/11 BND NXB XIC I:9.0/1 BND OTE O:16.0/11 EOR

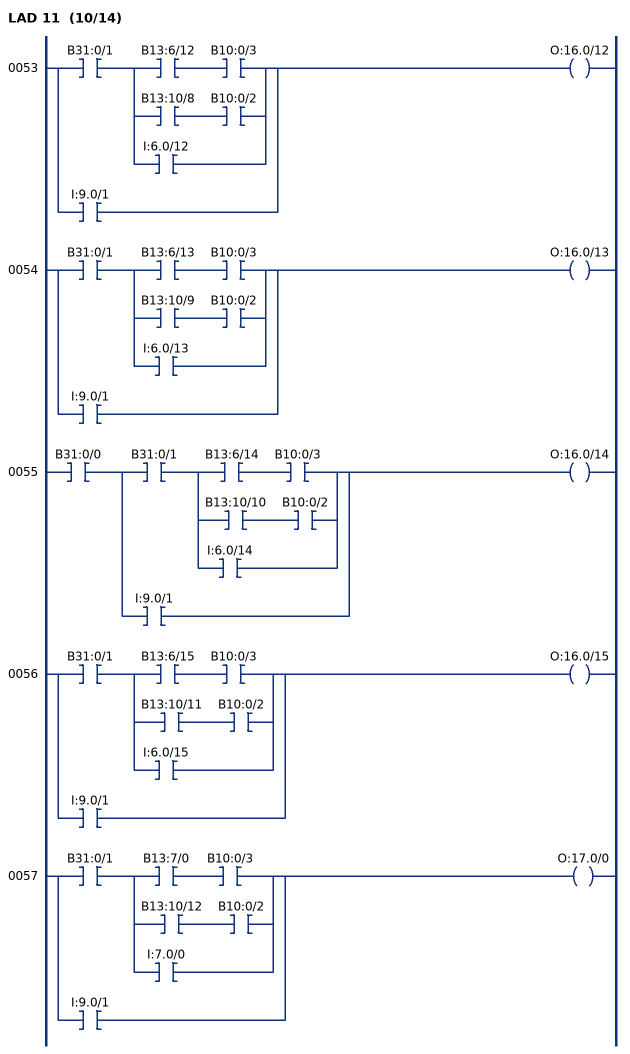
% Rung: 53 %
SOR BST XIC B31:0/1 BST XIC B13:6/12 XIC B10:0/3 NXB XIC B13:10/8 XIC B10:0/2 NXB XIC I:6.0/12 BND NXB XIC I:9.0/1 BND OTE O:16.0/12 EOR
% Rung: 54 %
SOR BST XIC B31:0/1 BST XIC B13:6/13 XIC B10:0/3 NXB XIC B13:10/9 XIC B10:0/2 NXB XIC I:6.0/13 BND NXB XIC I:9.0/1 BND OTE O:16.0/13 EOR
% Rung: 55 %
SOR XIC B31:0/0 BST XIC B31:0/1 BST XIC B13:6/14 XIC B10:0/3 NXB XIC B13:10/10 XIC B10:0/2 NXB XIC I:6.0/14 BND NXB XIC I:9.0/1 BND OTE O:16.0/14 EOR
% Rung: 56 %
SOR BST XIC B31:0/1 BST XIC B13:6/15 XIC B10:0/3 NXB XIC B13:10/11 XIC B10:0/2 NXB XIC I:6.0/15 BND NXB XIC I:9.0/1 BND OTE O:16.0/15 EOR
% Rung: 57 %
SOR BST XIC B31:0/1 BST XIC B13:7/0 XIC B10:0/3 NXB XIC B13:10/12 XIC B10:0/2 NXB XIC I:7.0/0 BND NXB XIC I:9.0/1 BND OTE O:17.0/0 EOR

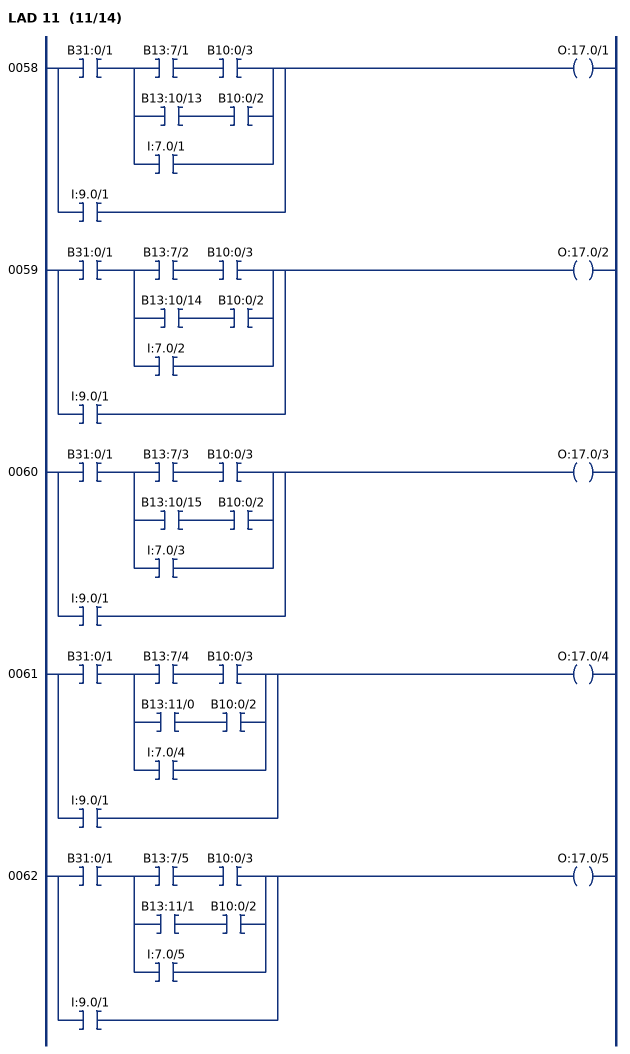
% Rung: 58 %
SOR BST XIC B31:0/1 BST XIC B13:7/1 XIC B10:0/3 NXB XIC B13:10/13 XIC B10:0/2 NXB XIC I:7.0/1 BND NXB XIC I:9.0/1 BND OTE O:17.0/1 EOR
% Rung: 59 %
SOR BST XIC B31:0/1 BST XIC B13:7/2 XIC B10:0/3 NXB XIC B13:10/14 XIC B10:0/2 NXB XIC I:7.0/2 BND NXB XIC I:9.0/1 BND OTE O:17.0/2 EOR
% Rung: 60 %
SOR BST XIC B31:0/1 BST XIC B13:7/3 XIC B10:0/3 NXB XIC B13:10/15 XIC B10:0/2 NXB XIC I:7.0/3 BND NXB XIC I:9.0/1 BND OTE O:17.0/3 EOR
% Rung: 61 %
SOR BST XIC B31:0/1 BST XIC B13:7/4 XIC B10:0/3 NXB XIC B13:11/0 XIC B10:0/2 NXB XIC I:7.0/4 BND NXB XIC I:9.0/1 BND OTE O:17.0/4 EOR
% Rung: 62 %
SOR BST XIC B31:0/1 BST XIC B13:7/5 XIC B10:0/3 NXB XIC B13:11/1 XIC B10:0/2 NXB XIC I:7.0/5 BND NXB XIC I:9.0/1 BND OTE O:17.0/5 EOR

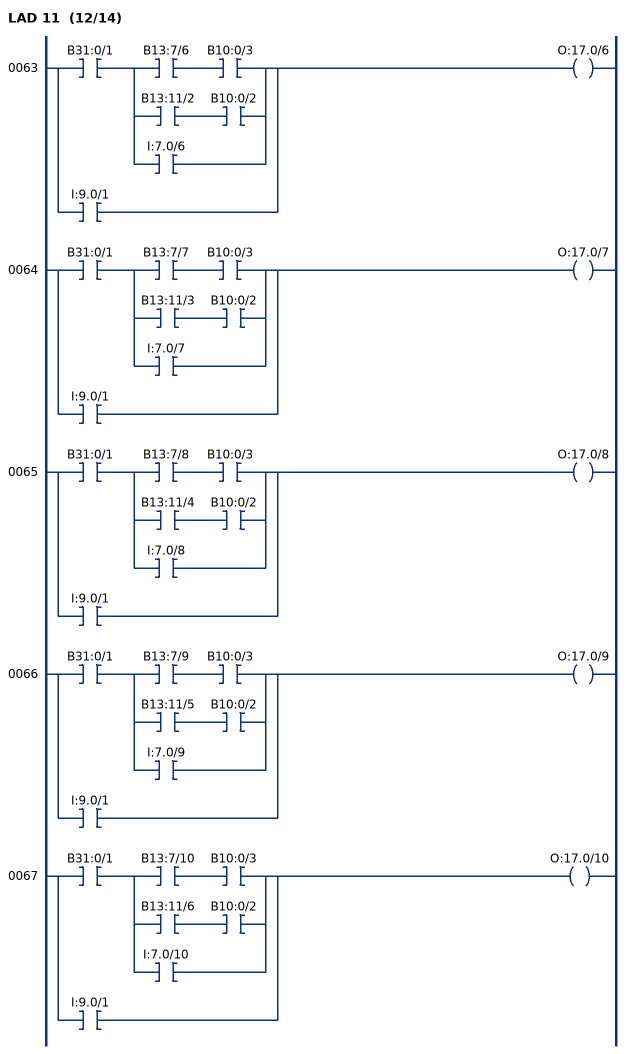
% Rung: 63 %
SOR BST XIC B31:0/1 BST XIC B13:7/6 XIC B10:0/3 NXB XIC B13:11/2 XIC B10:0/2 NXB XIC I:7.0/6 BND NXB XIC I:9.0/1 BND OTE O:17.0/6 EOR
% Rung: 64 %
SOR BST XIC B31:0/1 BST XIC B13:7/7 XIC B10:0/3 NXB XIC B13:11/3 XIC B10:0/2 NXB XIC I:7.0/7 BND NXB XIC I:9.0/1 BND OTE O:17.0/7 EOR
% Rung: 65 %
SOR BST XIC B31:0/1 BST XIC B13:7/8 XIC B10:0/3 NXB XIC B13:11/4 XIC B10:0/2 NXB XIC I:7.0/8 BND NXB XIC I:9.0/1 BND OTE O:17.0/8 EOR
% Rung: 66 %
SOR BST XIC B31:0/1 BST XIC B13:7/9 XIC B10:0/3 NXB XIC B13:11/5 XIC B10:0/2 NXB XIC I:7.0/9 BND NXB XIC I:9.0/1 BND OTE O:17.0/9 EOR
% Rung: 67 %
SOR BST XIC B31:0/1 BST XIC B13:7/10 XIC B10:0/3 NXB XIC B13:11/6 XIC B10:0/2 NXB XIC I:7.0/10 BND NXB XIC I:9.0/1 BND OTE O:17.0/10 EOR

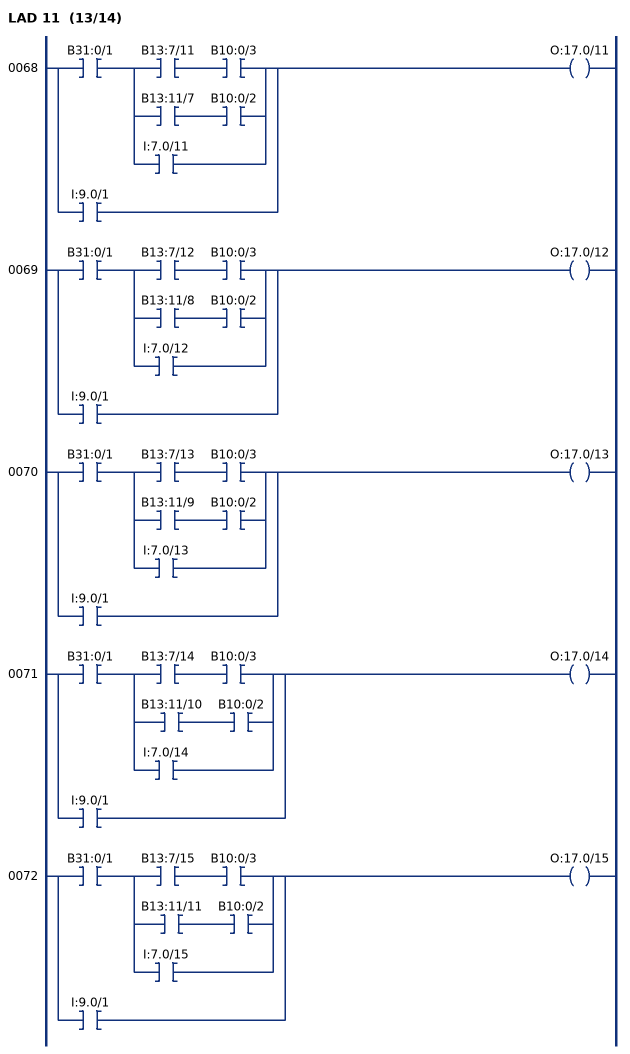
% Rung: 68 %
SOR BST XIC B31:0/1 BST XIC B13:7/11 XIC B10:0/3 NXB XIC B13:11/7 XIC B10:0/2 NXB XIC I:7.0/11 BND NXB XIC I:9.0/1 BND OTE O:17.0/11 EOR
% Rung: 69 %
SOR BST XIC B31:0/1 BST XIC B13:7/12 XIC B10:0/3 NXB XIC B13:11/8 XIC B10:0/2 NXB XIC I:7.0/12 BND NXB XIC I:9.0/1 BND OTE O:17.0/12 EOR
% Rung: 70 %
SOR BST XIC B31:0/1 BST XIC B13:7/13 XIC B10:0/3 NXB XIC B13:11/9 XIC B10:0/2 NXB XIC I:7.0/13 BND NXB XIC I:9.0/1 BND OTE O:17.0/13 EOR
% Rung: 71 %
SOR BST XIC B31:0/1 BST XIC B13:7/14 XIC B10:0/3 NXB XIC B13:11/10 XIC B10:0/2 NXB XIC I:7.0/14 BND NXB XIC I:9.0/1 BND OTE O:17.0/14 EOR
% Rung: 72 %
SOR BST XIC B31:0/1 BST XIC B13:7/15 XIC B10:0/3 NXB XIC B13:11/11 XIC B10:0/2 NXB XIC I:7.0/15 BND NXB XIC I:9.0/1 BND OTE O:17.0/15 EOR

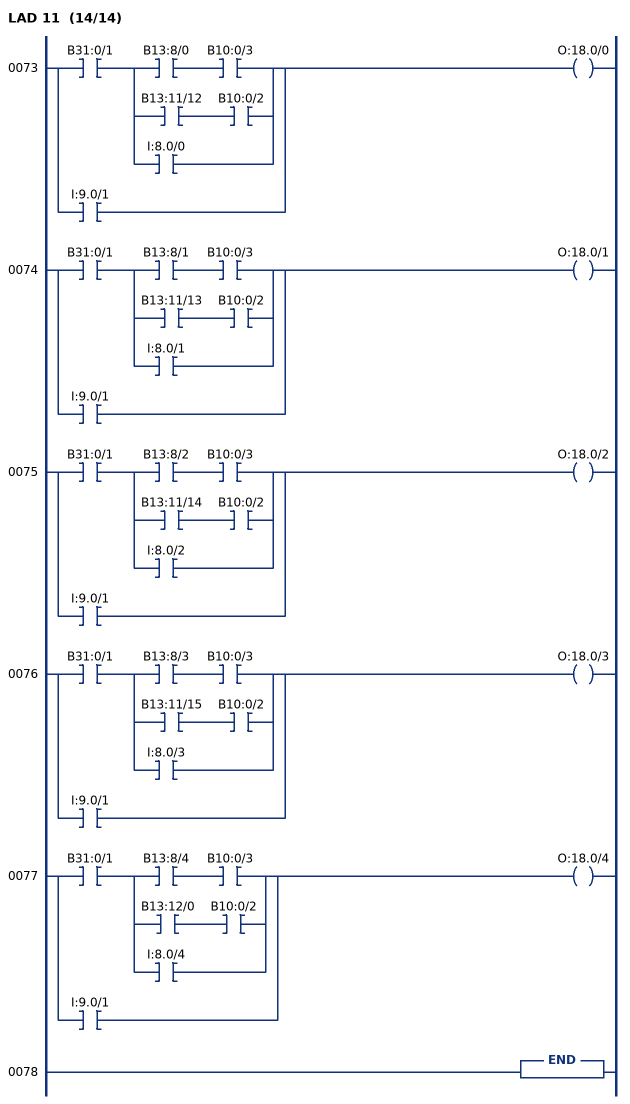
% Rung: 73 %
SOR BST XIC B31:0/1 BST XIC B13:8/0 XIC B10:0/3 NXB XIC B13:11/12 XIC B10:0/2 NXB XIC I:8.0/0 BND NXB XIC I:9.0/1 BND OTE O:18.0/0 EOR
% Rung: 74 %
SOR BST XIC B31:0/1 BST XIC B13:8/1 XIC B10:0/3 NXB XIC B13:11/13 XIC B10:0/2 NXB XIC I:8.0/1 BND NXB XIC I:9.0/1 BND OTE O:18.0/1 EOR
% Rung: 75 %
SOR BST XIC B31:0/1 BST XIC B13:8/2 XIC B10:0/3 NXB XIC B13:11/14 XIC B10:0/2 NXB XIC I:8.0/2 BND NXB XIC I:9.0/1 BND OTE O:18.0/2 EOR
% Rung: 76 %
SOR BST XIC B31:0/1 BST XIC B13:8/3 XIC B10:0/3 NXB XIC B13:11/15 XIC B10:0/2 NXB XIC I:8.0/3 BND NXB XIC I:9.0/1 BND OTE O:18.0/3 EOR
% Rung: 77 %
SOR BST XIC B31:0/1 BST XIC B13:8/4 XIC B10:0/3 NXB XIC B13:12/0 XIC B10:0/2 NXB XIC I:8.0/4 BND NXB XIC I:9.0/1 BND OTE O:18.0/4 EOR
% Rung: 78 %
SOR END EOR

DATA TABLE (non-zero values as saved)
DATA T11
% .PRE .ACC %
% T11:0 % 20 19
% T11:1 % 50 44
% T11:2 % 100 83
% T11:3 % 5 0
% T11:4 % 120 0
% T11:5 % 4 0
% T11:6 % 4 0
DATA T14
% .PRE .ACC %
% T14:1 % 2 0
% T14:2 % 5 0
% T14:3 % 5 0
% T14:4 % 5 0
% T14:5 % 5 0
% T14:6 % 5 0
% T14:7 % 5 0
% T14:8 % 5 0
% T14:9 % 5 0
% T14:10 % 5 0
% T14:11 % 5 0
% T14:12 % 5 0
% T14:13 % 5 0
% T14:14 % 5 0
% T14:15 % 5 0
% T14:16 % 5 0
% T14:17 % 5 0
% T14:18 % 5 0
% T14:19 % 5 0
% T14:20 % 5 0
% T14:21 % 5 0
% T14:22 % 5 0
% T14:23 % 5 0
% T14:24 % 5 0
% T14:25 % 5 0
% T14:26 % 5 0
% T14:27 % 5 0
% T14:28 % 5 0
% T14:29 % 5 0
% T14:30 % 5 0
% T14:31 % 5 0
% T14:32 % 5 0
% T14:33 % 5 0
% T14:34 % 5 0
% T14:35 % 5 0
% T14:36 % 5 0
% T14:37 % 5 0
% T14:38 % 5 0
% T14:39 % 5 0
% T14:40 % 5 0
% T14:41 % 5 0
% T14:42 % 5 0
% T14:43 % 5 0
% T14:44 % 5 0
% T14:45 % 5 0
% T14:46 % 5 0
% T14:47 % 5 0
% T14:48 % 5 0
% T14:49 % 5 0
% T14:50 % 5 0
% T14:51 % 5 0
% T14:52 % 5 0
% T14:53 % 5 0
% T14:54 % 5 0
% T14:55 % 5 0
% T14:56 % 5 0
% T14:57 % 5 0
% T14:58 % 5 0
% T14:59 % 5 0
DATA N15
% N15:0 % 16 0 0 0 0 0 0 0 0 0
DATA T17
% .PRE .ACC %
% T17:0 % 5 0
% T17:1 % 100 0
% T17:2 % 100 0
% T17:3 % 100 0
% T17:4 % 100 0
% T17:5 % 100 0
% T17:6 % 200 0
% T17:7 % 100 0
% T17:8 % 200 0
% T17:9 % 100 0
% T17:10 % 100 0
% T17:11 % 100 0
% T17:12 % 2000 0
% T17:13 % 100 0
% T17:14 % 100 0
% T17:15 % 100 0
% T17:16 % 500 0
% T17:17 % 100 0
% T17:18 % 100 0
% T17:19 % 100 0
% T17:20 % 100 0
% T17:21 % 100 0
% T17:22 % 100 0
% T17:23 % 300 0
% T17:24 % 100 0
% T17:25 % 100 0
% T17:26 % 100 0
% T17:27 % 100 0
% T17:28 % 100 0
% T17:29 % 100 0
% T17:30 % 100 0
% T17:31 % 100 0
% T17:32 % 100 0
% T17:33 % 100 0
% T17:34 % 2000 0
% T17:35 % 100 0
% T17:36 % 100 0
% T17:37 % 100 0
% T17:38 % 100 0
% T17:39 % 300 0
% T17:40 % 100 0
% T17:41 % 100 0
% T17:42 % 100 0
% T17:43 % 300 0
% T17:44 % 100 0
% T17:45 % 500 0
% T17:46 % 500 0
% T17:47 % 100 0
% T17:48 % 300 0
% T17:49 % 100 0
% T17:50 % 300 0
% T17:51 % 300 0
% T17:52 % 100 0
% T17:53 % 500 0
% T17:54 % 600 0
% T17:55 % 100 0
% T17:56 % 100 0
% T17:57 % 100 0
DATA T20
% .PRE .ACC %
% T20:0 % 5 0
% T20:1 % 100 0
% T20:2 % 100 0
% T20:3 % 100 0
% T20:4 % 100 0
% T20:5 % 100 0
% T20:6 % 100 0
% T20:7 % 100 0
% T20:8 % 100 0
% T20:9 % 100 0
% T20:10 % 100 0
% T20:11 % 1000 0
% T20:12 % 500 0
% T20:13 % 100 0
% T20:14 % 100 0
% T20:15 % 3000 0
% T20:16 % 100 0
% T20:17 % 100 0
% T20:18 % 100 0
% T20:19 % 100 0
% T20:20 % 100 0
% T20:21 % 100 0
% T20:22 % 100 0
% T20:23 % 100 0
% T20:24 % 100 0
% T20:25 % 100 0
% T20:26 % 500 0
% T20:27 % 400 0
% T20:28 % 400 0
% T20:29 % 100 0
% T20:30 % 100 0
% T20:31 % 100 0
% T20:32 % 100 0
% T20:33 % 500 0
% T20:34 % 100 0
% T20:35 % 100 0
% T20:36 % 100 0
% T20:37 % 100 0
% T20:38 % 100 0
% T20:39 % 100 0
% T20:40 % 100 0
% T20:41 % 3000 0
% T20:42 % 100 0
% T20:43 % 100 0
% T20:44 % 100 0
% T20:45 % 100 0
% T20:46 % 100 0
% T20:47 % 100 0
% T20:48 % 100 0
% T20:49 % 1000 0
% T20:50 % 100 0
% T20:51 % 100 0
% T20:52 % 1000 0
% T20:53 % 1000 0
% T20:54 % 500 0
% T20:55 % 100 0
% T20:56 % 100 0
% T20:57 % 2000 0
DATA T23
% .PRE .ACC %
% T23:0 % 5 0
% T23:1 % 25 0
% T23:2 % 25 0
% T23:3 % 500 0
% T23:4 % 25 0
% T23:5 % 100 0
% T23:6 % 25 0
% T23:7 % 1500 0
% T23:8 % 200 0
% T23:9 % 25 0
% T23:10 % 25 0
% T23:11 % 25 0
% T23:12 % 25 0
% T23:13 % 3 0
% T23:14 % 1000 0
% T23:15 % 300 0
% T23:16 % 120 0
DATA T26
% .PRE .ACC %
% T26:0 % 5 0
% T26:1 % 100 0
% T26:2 % 25 0
% T26:3 % 25 0
% T26:4 % 25 0
% T26:5 % 25 0
% T26:6 % 25 0
% T26:7 % 25 0
% T26:8 % 50 0
% T26:9 % 50 0
% T26:10 % 25 0
% T26:11 % 25 0
% T26:12 % 25 0
% T26:13 % 25 0
% T26:14 % 25 0
% T26:15 % 25 0
DATA T29
% .PRE .ACC %
% T29:0 % 50 50
% T29:1 % 50 50
